// Remet à a bonne échelle, map identique à celui d'arduino
FUNCTION MAP : LREAL
VAR_INPUT
	x : LREAL;
	in_min : LREAL;
	in_max : LREAL;
	out_min : LREAL;
	out_max : LREAL;
	
END_VAR
VAR
END_VAR


IF ((in_max - in_min) + out_min) <> 0 THEN
	MAP := (x - in_min) * (out_max - out_min) / (in_max - in_min) + out_min;
ELSE
	MAP := 0;
END_IF

RETURN;

END_FUNCTION

(* stored: Version 1.1.0.1, ProductVersion 3.1.4024.9
   POU MAP: Id {272632a0-ee8f-4a2e-adf4-67b985dedfce}, SpecialFunc None *)
